FUNCTION_BLOCK FB_HMI_ZNSE_ACTUATORS EXTENDS FB_HMI_COMPONENT
VAR_INPUT
END_VAR
VAR_OUTPUT
END_VAR
VAR
END_VAR
VAR_IN_OUT
	{attribute 'OPC.UA.DA' := '0'}
	fbInstance		: FB_NOTT_ZNSE_ACTUATORS;


END_VAR


fbHealthStatus( 
				bIsEnabled:= TRUE, 
				bIsGood := NOT fbInstance.stat.bError,
				bHasWarning := fbInstance.stat.bWarning
				);
				
fbBusyStatus(
				bIsBusy := fbInstance.stat.bBusy,
				bIsEnabled := TRUE);
				
M_UpdateStatusColor();

END_FUNCTION_BLOCK

(* stored: Version 1.1.0.1, ProductVersion 3.1.4024.14
   POU FB_HMI_ZNSE_ACTUATORS: Id {5d5e6c58-62c8-46d9-b2dc-67ab8ababe82}, SpecialFunc None *)
